TYPE E_SemiAutomatic :
(
	eSemi_ready := 0,
	eSemi_wayThere,
	eSemi_weld,
	eSemi_wayBack
);
END_TYPE

(* stored: Version 1.1.0.1
   DUT E_SemiAutomatic: Id {6e5c6811-3502-4ef3-b2c5-c4706872a56e} *)
